FUNCTION FC_NOT : BOOL
VAR_INPUT
	i:BOOL;
END_VAR
VAR
END_VAR

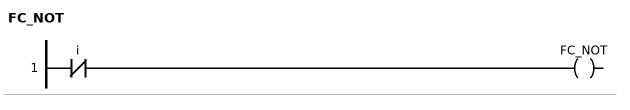
// NETWORK 1
FC_NOT := NOT i;

END_FUNCTION

(* stored: Version 1.1.0.1, ProductVersion 3.1.4024.11
   POU FC_NOT: Id {027cef92-e173-08d1-2a98-e6e0bb4baa84}, SpecialFunc None *)
